(* IEC 61131-3 sources: ATCMcontrol_Engineering/src/Target/ATHW119/Libs/ATCM_IEC1131_3, 218 files *)

(* ---- ABS.st ---- *)
(*[[
    UserURL= "ATCMfile:ABS.htm"
]]*)

FUNCTION ABS : any_num
VAR_INPUT
    IN : any_num;
END_VAR

overload lreal(lreal)
inline
{
	%1
	abs_lreal
}

overload real(real)
inline
{
	%1
	abs_real
}

overload dint(dint)
inline
{
	%1
	abs_dint
}

overload int(int)
inline
{
	%1
	abs_int
}

END_FUNCTION

(* ---- ACOS.st ---- *)
FUNCTION ACOS : any_real
VAR_INPUT
    IN : any_real;
END_VAR

overload lreal(lreal) inline { STDLIB(acos_lreal) }
overload real(real)   inline { STDLIB(acos_real) }

END_FUNCTION

(* ---- add.st ---- *)
(*[[
    UserURL= "ATCMFile:ADD.htm"
]]*)

FUNCTION ADD : ANY_MAGNITUDE
VAR_INPUT
    IN1 : ANY_MAGNITUDE;
END_VAR
VAR_IN_EXT
    IN2 : ANY_MAGNITUDE;
END_VAR

inline +

END_FUNCTION

(* ---- add_time.st ---- *)
(*[[
    UserURL= "ATCMfile:ADD_TIME.htm"
]]*)

FUNCTION ADD_TIME : TIME
VAR_INPUT
    IN1 : TIME;
    IN2 : TIME;
END_VAR

inline +

END_FUNCTION

(* ---- and.st ---- *)
(*[[
    UserURL= "ATCMfile:AND.htm"
]]*)

FUNCTION AND : ANY_BIT
VAR_INPUT
    IN1 : ANY_BIT;
END_VAR
VAR_IN_EXT
    IN2 : ANY_BIT;
END_VAR

inline AND

END_FUNCTION

(* ---- ASIN.st ---- *)
FUNCTION ASIN : any_real
VAR_INPUT
    IN : any_real;
END_VAR

overload lreal(lreal) inline { STDLIB(asin_lreal) }
overload real(real) inline   { STDLIB(asin_real) }

END_FUNCTION

(* ---- ATAN.st ---- *)
FUNCTION ATAN : any_real
VAR_INPUT
    IN : any_real;
END_VAR

overload lreal(lreal) inline { STDLIB(atan_lreal) }
overload real(real)   inline { STDLIB(atan_real) }

END_FUNCTION

(* ---- bool_to_byte.st ---- *)
(*[[
    UserURL= "ATCMfile:BOOL_TO_BYTE.htm"
]]*)

FUNCTION BOOL_TO_BYTE : BYTE
VAR_INPUT
    IN : BOOL;
END_VAR

inline { VMOP(bool_to_byte) }

END_FUNCTION

(* ---- bool_to_dint.st ---- *)
(*[[
    UserURL= "ATCMfile:BOOL_TO_DINT.htm"
]]*)

FUNCTION BOOL_TO_DINT : DINT
VAR_INPUT
    IN : BOOL;
END_VAR

inline{ VMOP(bool_to_dword) }

END_FUNCTION

(* ---- bool_to_dword.st ---- *)
(*[[
    UserURL= "ATCMfile:BOOL_TO_DWORD.htm"
]]*)

FUNCTION BOOL_TO_DWORD : DWORD
VAR_INPUT
    IN : BOOL;
END_VAR

inline{ VMOP(bool_to_dword) }

END_FUNCTION

(* ---- bool_to_int.st ---- *)
(*[[
    UserURL= "ATCMfile:BOOL_TO_DINT.htm"
]]*)

FUNCTION BOOL_TO_INT : INT
VAR_INPUT
    IN : BOOL;
END_VAR

inline{ VMOP(bool_to_word) }

END_FUNCTION

(* ---- bool_to_lreal.st ---- *)
(*[[
    UserURL= "ATCMfile:BOOL_TO_LREAL.htm"
]]*)

FUNCTION BOOL_TO_LREAL : LREAL
VAR_INPUT
    IN : BOOL;
END_VAR

inline{ VMOP(BOOL_TO_LREAL) }

END_FUNCTION

(* ---- bool_to_real.st ---- *)
(*[[
    UserURL= "ATCMfile:BOOL_TO_LREAL.htm"
]]*)

FUNCTION BOOL_TO_REAL : REAL
VAR_INPUT
    IN : BOOL;
END_VAR

inline{ VMOP }

END_FUNCTION

(* ---- bool_to_string.st ---- *)
(*[[
    UserURL= "ATCMfile:BOOL_TO_WSTRING.htm"
]]*)

FUNCTION BOOL_TO_STRING : STRING
VAR_INPUT
    IN : BOOL;
END_VAR

inline{ STDLIB(bool_to_string) }

END_FUNCTION

(* ---- bool_to_udint.st ---- *)
(*[[
    UserURL= "ATCMfile:BOOL_TO_UDINT.htm"
]]*)
FUNCTION BOOL_TO_UDINT : UDINT
VAR_INPUT
    IN : BOOL;
END_VAR

inline{ VMOP }

END_FUNCTION

(* ---- bool_to_uint.st ---- *)
(*[[
    UserURL= "ATCMfile:BOOL_TO_UINT.htm"
]]*)
FUNCTION BOOL_TO_UINT : UINT
VAR_INPUT
    IN : BOOL;
END_VAR

inline{ VMOP }

END_FUNCTION

(* ---- bool_to_word.st ---- *)
(*[[
    UserURL= "ATCMfile:BOOL_TO_WORD.htm"
]]*)

FUNCTION BOOL_TO_WORD : WORD
VAR_INPUT
    IN : BOOL;
END_VAR

inline{ VMOP }

END_FUNCTION

(* ---- byte_to_bool.st ---- *)
(*[[
    UserURL= "ATCMfile:BYTE_TO_BOOL.htm"
]]*)

FUNCTION BYTE_TO_BOOL : BOOL
VAR_INPUT
    IN : BYTE;
END_VAR

inline{VMOP}

END_FUNCTION

(* ---- byte_to_dint.st ---- *)
(*[[
    UserURL= "ATCMfile:BYTE_TO_DINT.htm"
]]*)

FUNCTION BYTE_TO_DINT : DINT
VAR_INPUT
    IN : BYTE;
END_VAR

inline{ VMOP(byte_to_dword) }

END_FUNCTION

(* ---- byte_to_dword.st ---- *)
(*[[
    UserURL= "ATCMfile:BYTE_TO_DWORD.htm"
]]*)

FUNCTION BYTE_TO_DWORD : DWORD
VAR_INPUT
    IN : BYTE;
END_VAR

inline{ VMOP }

END_FUNCTION

(* ---- byte_to_int.st ---- *)
(*[[
    UserURL= "ATCMfile:BYTE_TO_DINT.htm"
]]*)

FUNCTION BYTE_TO_INT : INT
VAR_INPUT
    IN : BYTE;
END_VAR

inline{ VMOP(byte_to_word) }

END_FUNCTION

(* ---- byte_to_lreal.st ---- *)
(*[[
    UserURL= "ATCMfile:BYTE_TO_LREAL.htm"
]]*)

FUNCTION BYTE_TO_LREAL : LREAL
VAR_INPUT
    IN : BYTE;
END_VAR

inline{VMOP}

END_FUNCTION

(* ---- byte_to_real.st ---- *)
(*[[
    UserURL= "ATCMfile:BYTE_TO_LREAL.htm"
]]*)

FUNCTION BYTE_TO_REAL : REAL
VAR_INPUT
    IN : BYTE;
END_VAR

inline{VMOP}

END_FUNCTION

(* ---- byte_to_string.st ---- *)
(*[[
    UserURL= "ATCMfile:BYTE_TO_WSTRING.htm"
]]*)

FUNCTION BYTE_TO_STRING : STRING
VAR_INPUT
    IN : BYTE;
END_VAR

inline{ STDLIB(byte_to_string) }

END_FUNCTION

(* ---- byte_to_udint.st ---- *)
(*[[
    UserURL= "ATCMfile:BYTE_TO_UDINT.htm"
]]*)
FUNCTION BYTE_TO_UDINT : UDINT
VAR_INPUT
    IN : BYTE;
END_VAR

inline{ VMOP }

END_FUNCTION

(* ---- byte_to_uint.st ---- *)
(*[[
    UserURL= "ATCMfile:BYTE_TO_UINT.htm"
]]*)
FUNCTION BYTE_TO_UINT : UINT
VAR_INPUT
    IN : BYTE;
END_VAR

inline{ VMOP }

END_FUNCTION

(* ---- byte_to_word.st ---- *)
(*[[
    UserURL= "ATCMfile:BYTE_TO_WORD.htm"
]]*)

FUNCTION BYTE_TO_WORD : WORD
VAR_INPUT
    IN : BYTE;
END_VAR

inline{VMOP}

END_FUNCTION

(* ---- CONCAT.st ---- *)
FUNCTION CONCAT : ANY_STRING
VAR_INPUT
    IN1 : ANY_STRING;
END_VAR
VAR_IN_EXT
    IN2 : ANY_STRING;
END_VAR

overload STRING(STRING,STRING,...) inline { STDLIB(ConcatString) }

END_FUNCTION

(* ---- COS.st ---- *)
FUNCTION COS : any_real
VAR_INPUT
    IN : any_real;
END_VAR

overload lreal(lreal) inline { STDLIB(cos_lreal) }
overload real(real) inline   { STDLIB(cos_real) }

END_FUNCTION

(* ---- DELETE.st ---- *)
FUNCTION DELETE : ANY_STRING
VAR_INPUT
    IN : ANY_STRING;
    L : ANY_INT;
    P : ANY_INT;
END_VAR

overload STRING(STRING,         INT,         INT) inline{ STDLIB(DeleteString_int)}
overload STRING(STRING, DINT to INT, DINT to INT) inline{ STDLIB(DeleteString_int)}

END_FUNCTION

(* ---- dint_to_bool.st ---- *)
(*[[
    UserURL= "ATCMfile:DINT_TO_BOOL.htm"
]]*)

FUNCTION DINT_TO_BOOL : BOOL
VAR_INPUT
    IN : DINT;
END_VAR

inline{ VMOP(dword_to_bool) }

END_FUNCTION

(* ---- dint_to_byte.st ---- *)
(*[[
    UserURL= "ATCMfile:DINT_TO_BYTE.htm"
]]*)

FUNCTION DINT_TO_BYTE : BYTE
VAR_INPUT
    IN : DINT;
END_VAR

inline{ VMOP }

END_FUNCTION

(* ---- dint_to_dword.st ---- *)
(*[[
    UserURL= "ATCMfile:DINT_TO_DWORD.htm"
]]*)

FUNCTION DINT_TO_DWORD : DWORD
VAR_INPUT
    IN : DINT;
END_VAR

inline{NOOP}

END_FUNCTION

(* ---- dint_to_int.st ---- *)
(*[[
    UserURL= "ATCMfile:DINT_TO_LINT.htm"
]]*)

FUNCTION DINT_TO_INT : INT
VAR_INPUT
    IN : DINT;
END_VAR

inline{VMOP}

END_FUNCTION

(* ---- dint_to_lreal.st ---- *)
(*[[
    UserURL= "ATCMfile:DINT_TO_LREAL.htm"
]]*)

FUNCTION DINT_TO_LREAL : LREAL
VAR_INPUT
    IN : DINT;
END_VAR

inline{VMOP}

END_FUNCTION

(* ---- dint_to_real.st ---- *)
(*[[
    UserURL= "ATCMfile:DINT_TO_LREAL.htm"
]]*)

FUNCTION DINT_TO_REAL : REAL
VAR_INPUT
    IN : DINT;
END_VAR

inline{VMOP}

END_FUNCTION

(* ---- dint_to_string.st ---- *)
(*[[
    UserURL= "ATCMfile:DINT_TO_WSTRING.htm"
]]*)

FUNCTION DINT_TO_STRING : STRING
VAR_INPUT
    IN : DINT;
END_VAR

inline{ STDLIB(dint_to_string) }

END_FUNCTION

(* ---- dint_to_time.st ---- *)
(*[[
    UserURL= "ATCMfile:DINT_TO_TIME.htm"
]]*)

FUNCTION DINT_TO_TIME : TIME
VAR_INPUT
    IN : DINT;
END_VAR

inline { %1 }

END_FUNCTION

(* ---- dint_to_udint.st ---- *)
(*[[
    UserURL= "ATCMfile:DINT_TO_UDINT.htm"
]]*)
FUNCTION DINT_TO_UDINT : UDINT
VAR_INPUT
    IN : DINT;
END_VAR

inline{NOOP}

END_FUNCTION

(* ---- dint_to_uint.st ---- *)
(*[[
    UserURL= "ATCMfile:DINT_TO_UINT.htm"
]]*)
FUNCTION DINT_TO_UINT : UINT
VAR_INPUT
    IN : DINT;
END_VAR

inline{ VMOP }

END_FUNCTION

(* ---- dint_to_word.st ---- *)
(*[[
    UserURL= "ATCMfile:DINT_TO_WORD.htm"
]]*)

FUNCTION DINT_TO_WORD : WORD
VAR_INPUT
    IN : DINT;
END_VAR

inline{VMOP}

END_FUNCTION

(* ---- div.st ---- *)
(*[[
    UserURL= "ATCMfile:DIV.htm"
]]*)

FUNCTION DIV : ANY_NUM
VAR_INPUT
    IN1: ANY_NUM;
    IN2: ANY_NUM;
END_VAR

inline /

END_FUNCTION

(* ---- divtime.st ---- *)
(*[[
    UserURL= "ATCMfile:DIVTIME.htm"
]]*)

FUNCTION DIVTIME : TIME
VAR_INPUT
    IN1 : TIME;
    IN2 : ANY_NUM;
END_VAR

overload TIME(TIME,INT)
inline
{
    %1
    %2
    int_to_dint
    div_dint
}

overload TIME(TIME,DINT)
inline
{
    %1
    %2
    div_dint
}

overload TIME(TIME,REAL)
inline
{
    %1
    dint_to_real
    %2
    div_real
    real_to_dint
}

overload TIME(TIME,LREAL)
inline
{
    %1
    dint_to_lreal
    %2
    div_lreal
    lreal_to_dint
}

END_FUNCTION

(* ---- dword_to_bool.st ---- *)
(*[[
    UserURL= "ATCMfile:DWORD_TO_BOOL.htm"
]]*)

FUNCTION DWORD_TO_BOOL : BOOL
VAR_INPUT
    IN : DWORD;
END_VAR

inline{VMOP}

END_FUNCTION

(* ---- dword_to_byte.st ---- *)
(*[[
    UserURL= "ATCMfile:DWORD_TO_BYTE.htm"
]]*)

FUNCTION DWORD_TO_BYTE : BYTE
VAR_INPUT
    IN : DWORD;
END_VAR

inline{VMOP}

END_FUNCTION

(* ---- dword_to_dint.st ---- *)
(*[[
    UserURL= "ATCMfile:DWORD_TO_DINT.htm"
]]*)

FUNCTION DWORD_TO_DINT : DINT
VAR_INPUT
    IN : DWORD;
END_VAR

inline{VMOP}

END_FUNCTION

(* ---- dword_to_int.st ---- *)
(*[[
    UserURL= "ATCMfile:DWORD_TO_LINT.htm"
]]*)

FUNCTION DWORD_TO_INT : INT
VAR_INPUT
    IN : DWORD;
END_VAR

inline{VMOP}

END_FUNCTION

(* ---- dword_to_lreal.st ---- *)
(*[[
    UserURL= "ATCMfile:DWORD_TO_LREAL.htm"
]]*)

FUNCTION DWORD_TO_LREAL : LREAL
VAR_INPUT
    IN : DWORD;
END_VAR

inline{VMOP}

END_FUNCTION

(* ---- dword_to_lword.st ---- *)
(*[[
    UserURL= "ATCMfile:DWORD_TO_LWORD.htm"
]]*)

FUNCTION DWORD_TO_LWORD : LWORD
VAR_INPUT
    IN : DWORD;
END_VAR

inline{VMOP}

END_FUNCTION

(* ---- dword_to_real.st ---- *)
(*[[
    UserURL= "ATCMfile:DWORD_TO_LREAL.htm"
]]*)

FUNCTION DWORD_TO_REAL : REAL
VAR_INPUT
    IN : DWORD;
END_VAR

inline{VMOP}

END_FUNCTION

(* ---- dword_to_string.st ---- *)
(*[[
    UserURL= "ATCMfile:DWORD_TO_WSTRING.htm"
]]*)

FUNCTION DWORD_TO_STRING : STRING
VAR_INPUT
    IN : DWORD;
END_VAR

inline{ STDLIB(dword_to_string) }

END_FUNCTION

(* ---- dword_to_udint.st ---- *)
(*[[
    UserURL= "ATCMfile:DWORD_TO_UDINT.htm"
]]*)
FUNCTION DWORD_TO_UDINT : UDINT
VAR_INPUT
    IN : DWORD;
END_VAR

inline{NOOP}

END_FUNCTION

(* ---- dword_to_uint.st ---- *)
(*[[
    UserURL= "ATCMfile:DWORD_TO_UINT.htm"
]]*)
FUNCTION DWORD_TO_UINT : UINT
VAR_INPUT
    IN : DWORD;
END_VAR

inline{ VMOP }

END_FUNCTION

(* ---- dword_to_word.st ---- *)
(*[[
    UserURL= "ATCMfile:DWORD_TO_WORD.htm"
]]*)

FUNCTION DWORD_TO_WORD : WORD
VAR_INPUT
    IN : DWORD;
END_VAR

inline{VMOP(dword_to_uint)}

END_FUNCTION

(* ---- eq.st ---- *)
(*[[
    UserURL= "ATCMfile:EQ.htm"
]]*)

FUNCTION EQ : BOOL
VAR_INPUT
    IN1 : ANY_ELEMENTARY;
END_VAR
VAR_IN_EXT
    IN2 : ANY_ELEMENTARY;
END_VAR

inline =

END_FUNCTION

(* ---- EXP.st ---- *)
FUNCTION EXP : any_real
VAR_INPUT
    IN : any_real;
END_VAR

overload lreal(lreal) inline { STDLIB(exp_lreal) }
overload real(real)   inline { STDLIB(exp_real) }

END_FUNCTION

(* ---- expt.st ---- *)
(*[[
    UserURL= "ATCMfile:EXPT.htm"
]]*)

FUNCTION EXPT : ANY_REAL
VAR_INPUT
    IN1: ANY_REAL;
    IN2: ANY_NUM;
END_VAR

overload REAL(REAL,DINT)    inline
{
    %1
    %2
    pow_real_dint
}
overload REAL(REAL,INT)     inline
{
    %1
    %2
    pow_real_int
}
overload LREAL(LREAL,DINT)  inline
{
    %1
    %2
    pow_lreal_dint
}
overload LREAL(LREAL,INT)   inline
{
    %1
    %2
    pow_lreal_int
}
overload REAL(REAL,REAL)    inline
{
    %1
    %2
    pow_real_real
}
overload LREAL(LREAL,LREAL) inline
{
    %1
    %2
    pow_lreal_lreal
}
overload REAL(REAL,LREAL)   inline
{
    %1
    real_to_lreal
    %2
    pow_lreal_lreal
    lreal_to_real
}
overload LREAL(LREAL,REAL)  inline
{
    %1
    %2
    real_to_lreal
    pow_lreal_lreal
}

END_FUNCTION

(* ---- FIND.st ---- *)
FUNCTION FIND : ANY_INT
VAR_INPUT
    IN1 : ANY_STRING;
    IN2 : ANY_STRING;
END_VAR

overload INT        (STRING, STRING) inline{ STDLIB(FindString_int) }
overload INT to DINT(STRING, STRING) inline{ STDLIB(FindString_int) }

END_FUNCTION

(* ---- ge.st ---- *)
(*[[
    UserURL= "ATCMfile:GE.htm"
]]*)

FUNCTION GE : BOOL
VAR_INPUT
    IN1 : ANY_ELEMENTARY;
END_VAR
VAR_IN_EXT
    IN2 : ANY_ELEMENTARY;
END_VAR

inline >=

END_FUNCTION

(* ---- gt.st ---- *)
(*[[
    UserURL= "ATCMfile:GT.htm"
]]*)

FUNCTION GT : BOOL
VAR_INPUT
    IN1 : ANY_ELEMENTARY;
END_VAR
VAR_IN_EXT
    IN2 : ANY_ELEMENTARY;
END_VAR

inline >

END_FUNCTION

(* ---- INSERT.st ---- *)
FUNCTION INSERT : ANY_STRING
VAR_INPUT
    IN1 : ANY_STRING;
    IN2 : ANY_STRING;
    P : ANY_INT;
END_VAR

overload STRING(STRING, STRING,         INT) inline{ STDLIB(InsertString_int)}
overload STRING(STRING, STRING, DINT to INT) inline{ STDLIB(InsertString_int)}

END_FUNCTION

(* ---- int_to_bool.st ---- *)
(*[[
    UserURL= "ATCMfile:DINT_TO_BOOL.htm"
]]*)

FUNCTION INT_TO_BOOL : BOOL
VAR_INPUT
    IN : INT;
END_VAR

inline{VMOP(WORD_TO_BOOL)}

END_FUNCTION

(* ---- int_to_byte.st ---- *)
(*[[
    UserURL= "ATCMfile:DINT_TO_BYTE.htm"
]]*)

FUNCTION INT_TO_BYTE : BYTE
VAR_INPUT
    IN : INT;
END_VAR

inline{VMOP(word_to_byte)}

END_FUNCTION

(* ---- int_to_dint.st ---- *)
(*[[
    UserURL= "ATCMfile:DINT_TO_LINT.htm"
]]*)

FUNCTION INT_TO_DINT : DINT
VAR_INPUT
    IN : INT;
END_VAR

inline{VMOP}

END_FUNCTION

(* ---- int_to_dword.st ---- *)
(*[[
    UserURL= "ATCMfile:DINT_TO_DWORD.htm"
]]*)

FUNCTION INT_TO_DWORD : DWORD
VAR_INPUT
    IN : INT;
END_VAR

inline{VMOP(int_to_dword)}

END_FUNCTION

(* ---- int_to_lint.st ---- *)
(*[[
    UserURL= "ATCMfile:DINT_TO_LINT.htm"
]]*)

FUNCTION INT_TO_LINT : LINT
VAR_INPUT
    IN : INT;
END_VAR

inline{VMOP}

END_FUNCTION

(* ---- int_to_lreal.st ---- *)
(*[[
    UserURL= "ATCMfile:DINT_TO_LREAL.htm"
]]*)

FUNCTION INT_TO_LREAL : LREAL
VAR_INPUT
    IN : INT;
END_VAR

inline{VMOP}

END_FUNCTION

(* ---- int_to_real.st ---- *)
(*[[
    UserURL= "ATCMfile:DINT_TO_LREAL.htm"
]]*)

FUNCTION INT_TO_REAL : REAL
VAR_INPUT
    IN : INT;
END_VAR

inline{VMOP}

END_FUNCTION

(* ---- int_to_string.st ---- *)
(*[[
    UserURL= "ATCMfile:DINT_TO_WSTRING.htm"
]]*)

FUNCTION INT_TO_STRING : STRING
VAR_INPUT
    IN : INT;
END_VAR

inline{ STDLIB(int_to_string) }

END_FUNCTION

(* ---- int_to_time.st ---- *)
(*[[
    UserURL= "ATCMfile:DINT_TO_TIME.htm"
]]*)

FUNCTION INT_TO_TIME : TIME
VAR_INPUT
    IN : INT;
END_VAR

inline
{
	%1
	int_to_dint
}

END_FUNCTION

(* ---- int_to_udint.st ---- *)
(*[[
    UserURL= "ATCMfile:INT_TO_UDINT.htm"
]]*)
FUNCTION INT_TO_UDINT : UDINT
VAR_INPUT
    IN : INT;
END_VAR

inline{ VMOP }

END_FUNCTION

(* ---- int_to_uint.st ---- *)
(*[[
    UserURL= "ATCMfile:INT_TO_UINT.htm"
]]*)
FUNCTION INT_TO_UINT : UINT
VAR_INPUT
    IN : INT;
END_VAR

inline{NOOP}

END_FUNCTION

(* ---- int_to_word.st ---- *)
(*[[
    UserURL= "ATCMfile:DINT_TO_WORD.htm"
]]*)

FUNCTION INT_TO_WORD : WORD
VAR_INPUT
    IN : INT;
END_VAR

inline{NOOP}

END_FUNCTION

(* ---- le.st ---- *)
(*[[
    UserURL= "ATCMfile:LE.htm"
]]*)

FUNCTION LE : BOOL
VAR_INPUT
    IN1 : ANY_ELEMENTARY;
END_VAR
VAR_IN_EXT
    IN2 : ANY_ELEMENTARY;
END_VAR

inline <=

END_FUNCTION

(* ---- LEFT.st ---- *)
FUNCTION LEFT : ANY_STRING
VAR_INPUT
    IN : ANY_STRING;
    L : ANY_INT;
END_VAR

overload STRING(STRING, INT)          inline{ STDLIB(LeftString_int) }
overload STRING(STRING, DINT to INT)  inline{ STDLIB(LeftString_int) }

END_FUNCTION

(* ---- LEN.st ---- *)
FUNCTION LEN : ANY_INT
VAR_INPUT
    IN : STRING;
END_VAR

overload INT        (STRING) inline { STDLIB(strlen_int) }
overload INT to DINT(STRING) inline { STDLIB(strlen_int) }

END_FUNCTION

(* ---- limit.st ---- *)
(*[[
    UserURL= "ATCMfile:LIMIT.htm"
]]*)

FUNCTION LIMIT : ANY_ELEMENTARY
VAR_INPUT
    MN : ANY_ELEMENTARY;
    IN : ANY_ELEMENTARY;
    MX : ANY_ELEMENTARY;
END_VAR

overload BOOL(BOOL,BOOL,BOOL) inline
{
    %2
    %1
    or_bool
    %3
    and_bool
}
overload BYTE(BYTE, BYTE, BYTE) inline
{
    %2
    %1
    lt_byte
    jmpcn L1%u
    %1
    jmp Lend%u
:L1%u
    %2
    %3
    gt_byte
    jmpcn L2%u
    %3
    jmp Lend%u
:L2%u
    %2
:Lend%u
}
overload WORD(WORD, WORD, WORD) inline
{
    %2
    %1
    lt_word
    jmpcn L1%u
    %1
    jmp Lend%u
:L1%u
    %2
    %3
    gt_word
    jmpcn L2%u
    %3
    jmp Lend%u
:L2%u
    %2
:Lend%u
}
overload DWORD(DWORD, DWORD, DWORD) inline
{
    %2
    %1
    lt_dword
    jmpcn L1%u
    %1
    jmp Lend%u
:L1%u
    %2
    %3
    gt_dword
    jmpcn L2%u
    %3
    jmp Lend%u
:L2%u
    %2
:Lend%u
}
overload INT(INT, INT, INT) inline
{
    %2
    %1
    lt_int
    jmpcn L1%u
    %1
    jmp Lend%u
:L1%u
    %2
    %3
    gt_int
    jmpcn L2%u
    %3
    jmp Lend%u
:L2%u
    %2
:Lend%u
}
overload DINT|TIME(DINT|TIME, DINT|TIME, DINT|TIME) inline
{
    %2
    %1
    lt_dint
    jmpcn L1%u
    %1
    jmp Lend%u
:L1%u
    %2
    %3
    gt_dint
    jmpcn L2%u
    %3
    jmp Lend%u
:L2%u
    %2
:Lend%u
}
overload REAL(REAL,REAL,REAL) inline
{
    %2
    %1
    lt_real
    jmpcn L1%u
    %1
    jmp Lend%u
:L1%u
    %2
    %3
    gt_real
    jmpcn L2%u
    %3
    jmp Lend%u
:L2%u
    %2
:Lend%u
}

overload LREAL(LREAL,LREAL,LREAL) inline
{
    %2
    %1
    lt_lreal
    jmpcn L1%u
    %1
    jmp Lend%u
:L1%u
    %2
    %3
    gt_lreal
    jmpcn L2%u
    %3
    jmp Lend%u
:L2%u
    %2
:Lend%u
}

overload STRING(STRING, STRING, STRING) inline
{
    %2
    %1
    lt_string
    jmpcn L1%u
    %1
    jmp Lend%u
:L1%u
    %2
    %3
    gt_string
    jmpcn L2%u
    %3
    jmp Lend%u
:L2%u
    %2
:Lend%u
}

END_FUNCTION

(* ---- lint_to_bool.st ---- *)
(*[[
    UserURL= "ATCMfile:LINT_TO_BOOL.htm"
]]*)

FUNCTION LINT_TO_BOOL : BOOL
VAR_INPUT
    IN : LINT;
END_VAR

inline{%1==0l?false:true}

END_FUNCTION

(* ---- lint_to_byte.st ---- *)
(*[[
    UserURL= "ATCMfile:LINT_TO_BYTE.htm"
]]*)

FUNCTION LINT_TO_BYTE : BYTE
VAR_INPUT
    IN : LINT;
END_VAR

inline{(int)%1&0xff}

END_FUNCTION

(* ---- lint_to_dint.st ---- *)
(*[[
    UserURL= "ATCMfile:LINT_TO_DINT.htm"
]]*)

FUNCTION LINT_TO_DINT : DINT
VAR_INPUT
    IN : LINT;
END_VAR

inline{(int)%1}

END_FUNCTION

(* ---- lint_to_dword.st ---- *)
(*[[
    UserURL= "ATCMfile:LINT_TO_DWORD.htm"
]]*)

FUNCTION LINT_TO_DWORD : DWORD
VAR_INPUT
    IN : LINT;
END_VAR

inline{(int)%1}

END_FUNCTION

(* ---- lint_to_int.st ---- *)
(*[[
    UserURL= "ATCMfile:LINT_TO_DINT.htm"
]]*)

FUNCTION LINT_TO_INT : INT
VAR_INPUT
    IN : LINT;
END_VAR

inline{(int)%1}

END_FUNCTION

(* ---- lint_to_lreal.st ---- *)
(*[[
    UserURL= "ATCMfile:LINT_TO_LREAL.htm"
]]*)

FUNCTION LINT_TO_LREAL : LREAL
VAR_INPUT
    IN : LINT;
END_VAR

inline{(double)%1}

END_FUNCTION

(* ---- lint_to_lword.st ---- *)
(*[[
    UserURL= "ATCMfile:LINT_TO_LWORD.htm"
]]*)

FUNCTION LINT_TO_LWORD : LWORD
VAR_INPUT
    IN : LINT;
END_VAR

inline{%1}

END_FUNCTION

(* ---- lint_to_real.st ---- *)
(*[[
    UserURL= "ATCMfile:LINT_TO_LREAL.htm"
]]*)

FUNCTION LINT_TO_REAL : REAL
VAR_INPUT
    IN : LINT;
END_VAR

inline{(double)%1}

END_FUNCTION

(* ---- lint_to_string.st ---- *)
(*[[
    UserURL= "ATCMfile:LINT_TO_WSTRING.htm"
]]*)

FUNCTION LINT_TO_STRING : STRING
VAR_INPUT
    IN : LINT;
END_VAR

inline{java.lang.Long.toString(%1)}

END_FUNCTION

(* ---- lint_to_time.st ---- *)
(*[[
    UserURL= "ATCMfile:LINT_TO_TIME.htm"
]]*)

FUNCTION LINT_TO_TIME : TIME
VAR_INPUT
    IN : LINT;
END_VAR

inline{%1}

END_FUNCTION

(* ---- lint_to_word.st ---- *)
(*[[
    UserURL= "ATCMfile:LINT_TO_WORD.htm"
]]*)

FUNCTION LINT_TO_WORD : WORD
VAR_INPUT
    IN : LINT;
END_VAR

inline{(int)%1&0xffff}

END_FUNCTION

(* ---- LN.st ---- *)
FUNCTION LN : any_real
VAR_INPUT
    IN : any_real;
END_VAR

overload lreal(lreal) inline { STDLIB(log_lreal) }
overload real(real)   inline { STDLIB(log_real) }

END_FUNCTION

(* ---- LOG.st ---- *)
FUNCTION LOG : any_real
VAR_INPUT
    IN : any_real;
END_VAR

overload lreal(lreal) inline { STDLIB(log10_lreal) }
overload real(real)   inline { STDLIB(log10_real) }

END_FUNCTION

(* ---- lreal_to_bool.st ---- *)
(*[[
    UserURL= "ATCMfile:LREAL_TO_BOOL.htm"
]]*)

FUNCTION LREAL_TO_BOOL : BOOL
VAR_INPUT
    IN : LREAL;
END_VAR

inline{VMOP}

END_FUNCTION

(* ---- lreal_to_byte.st ---- *)
(*[[
    UserURL= "ATCMfile:LREAL_TO_BYTE.htm"
]]*)

FUNCTION LREAL_TO_BYTE : BYTE
VAR_INPUT
    IN : LREAL;
END_VAR

inline{VMOP}

END_FUNCTION

(* ---- lreal_to_dint.st ---- *)
(*[[
    UserURL= "ATCMfile:LREAL_TO_DINT.htm"
]]*)

FUNCTION LREAL_TO_DINT : DINT
VAR_INPUT
    IN : LREAL;
END_VAR

inline{VMOP}

END_FUNCTION

(* ---- lreal_to_dword.st ---- *)
(*[[
    UserURL= "ATCMfile:LREAL_TO_DWORD.htm"
]]*)

FUNCTION LREAL_TO_DWORD : DWORD
VAR_INPUT
    IN : LREAL;
END_VAR

inline{VMOP}

END_FUNCTION

(* ---- lreal_to_int.st ---- *)
(*[[
    UserURL= "ATCMfile:LREAL_TO_LINT.htm"
]]*)

FUNCTION LREAL_TO_INT : INT
VAR_INPUT
    IN : LREAL;
END_VAR

inline{VMOP}

END_FUNCTION

(* ---- lreal_to_lint.st ---- *)
(*[[
    UserURL= "ATCMfile:LREAL_TO_LINT.htm"
]]*)

FUNCTION LREAL_TO_LINT : LINT
VAR_INPUT
    IN : LREAL;
END_VAR

inline{VMOP(not_yet_implem)}

END_FUNCTION

(* ---- lreal_to_lword.st ---- *)
(*
 * Note:
 *  LREAL_TO_LWORD(x) is the same as
 *  LINT_TO_LWORD(LREAL_TO_LINT(x))
 *
 *  e.g.  LREAL_TO_LWORD(-1.0E0) = 16#ffffffffffffffff;
 *)

FUNCTION LREAL_TO_LWORD : LWORD
VAR_INPUT
    IN : LREAL;
END_VAR

inline{VMOP(not_yet_implem)}

END_FUNCTION

(* ---- lreal_to_real.st ---- *)
(*[[
    UserURL= "ATCMfile:LREAL_TO_TIME.htm"
]]*)

FUNCTION LREAL_TO_REAL : REAL
VAR_INPUT
    IN : LREAL;
END_VAR

inline{VMOP}

END_FUNCTION

(* ---- lreal_to_string.st ---- *)
(*[[
    UserURL= "ATCMfile:LREAL_TO_WSTRING.htm"
]]*)

FUNCTION LREAL_TO_STRING : STRING
VAR_INPUT
    IN : LREAL;
END_VAR

inline{ STDLIB(lreal_to_string)}

END_FUNCTION

(* ---- lreal_to_time.st ---- *)
(*[[
    UserURL= "ATCMfile:LREAL_TO_TIME.htm"
]]*)

FUNCTION LREAL_TO_TIME : TIME
VAR_INPUT
    IN : LREAL;
END_VAR

inline
{
    %1
	lreal_to_dint
}

END_FUNCTION

(* ---- lreal_to_udint.st ---- *)
(*[[
    UserURL= "ATCMfile:LREAL_TO_UDINT.htm"
]]*)
FUNCTION LREAL_TO_UDINT : UDINT
VAR_INPUT
    IN : LREAL;
END_VAR

inline{ VMOP }

END_FUNCTION

(* ---- lreal_to_uint.st ---- *)
(*[[
    UserURL= "ATCMfile:LREAL_TO_UINT.htm"
]]*)
FUNCTION LREAL_TO_UINT : UINT
VAR_INPUT
    IN : LREAL;
END_VAR

inline{ VMOP }

END_FUNCTION

(* ---- lreal_to_word.st ---- *)
(*[[
    UserURL= "ATCMfile:LREAL_TO_WORD.htm"
]]*)

FUNCTION LREAL_TO_WORD : WORD
VAR_INPUT
    IN : LREAL;
END_VAR

inline{VMOP}

END_FUNCTION

(* ---- lt.st ---- *)
(*[[
    UserURL= "ATCMfile:LT.htm"
]]*)

FUNCTION LT : BOOL
VAR_INPUT
    IN1 : ANY_ELEMENTARY;
END_VAR
VAR_IN_EXT
    IN2 : ANY_ELEMENTARY;
END_VAR

inline <

END_FUNCTION

(* ---- lword_to_bool.st ---- *)
(*[[
    UserURL= "ATCMfile:LWORD_TO_BOOL.htm"
]]*)

FUNCTION LWORD_TO_BOOL : BOOL
VAR_INPUT
    IN : LWORD;
END_VAR

inline{%1==0l?false:true}

END_FUNCTION

(* ---- lword_to_byte.st ---- *)
(*[[
    UserURL= "ATCMfile:LWORD_TO_BYTE.htm"
]]*)

FUNCTION LWORD_TO_BYTE : BYTE
VAR_INPUT
    IN : LWORD;
END_VAR

inline{(int)%1&0xff}

END_FUNCTION

(* ---- lword_to_dint.st ---- *)
(*[[
    UserURL= "ATCMfile:LWORD_TO_DINT.htm"
]]*)

FUNCTION LWORD_TO_DINT : DINT
VAR_INPUT
    IN : LWORD;
END_VAR

inline{(int)%1}

END_FUNCTION

(* ---- lword_to_dword.st ---- *)
(*[[
    UserURL= "ATCMfile:LWORD_TO_DWORD.htm"
]]*)

FUNCTION LWORD_TO_DWORD : DWORD
VAR_INPUT
    IN : LWORD;
END_VAR

inline{(int)%1}

END_FUNCTION

(* ---- lword_to_int.st ---- *)
(*[[
    UserURL= "ATCMfile:LWORD_TO_DINT.htm"
]]*)

FUNCTION LWORD_TO_INT : INT
VAR_INPUT
    IN : LWORD;
END_VAR

inline{(int)%1}

END_FUNCTION

(* ---- lword_to_lint.st ---- *)
(*[[
    UserURL= "ATCMfile:LWORD_TO_LINT.htm"
]]*)

FUNCTION LWORD_TO_LINT : LINT
VAR_INPUT
    IN : LWORD;
END_VAR

inline{%1}

END_FUNCTION

(* ---- lword_to_lreal.st ---- *)
(*
 * Note:
 *  LWORD_TO_LREAL(x) is the same as
 *  LINT_TO_LREAL(LWORD_TO_LINT(x))
 *
 *  e.g.  LWORD_TO_LREAL(16#ffffffffffffffff) = -1.0E0
 *)
FUNCTION LWORD_TO_LREAL : LREAL
VAR_INPUT
    IN : LWORD;
END_VAR

inline{(double)%1}

END_FUNCTION

(* ---- lword_to_real.st ---- *)
(*
 * Note:
 *  LWORD_TO_LREAL(x) is the same as
 *  LINT_TO_LREAL(LWORD_TO_LINT(x))
 *
 *  e.g.  LWORD_TO_LREAL(16#ffffffffffffffff) = -1.0E0
 *)
FUNCTION LWORD_TO_REAL : REAL
VAR_INPUT
    IN : LWORD;
END_VAR

inline{(double)%1}

END_FUNCTION

(* ---- lword_to_string.st ---- *)
(*[[
    UserURL= "ATCMfile:LWORD_TO_WSTRING.htm"
]]*)

FUNCTION LWORD_TO_STRING : STRING
VAR_INPUT
    IN : LWORD;
END_VAR

inline{ STDLIB(not yet implemented) }

END_FUNCTION

(* ---- lword_to_word.st ---- *)
(*[[
    UserURL= "ATCMfile:LWORD_TO_WORD.htm"
]]*)

FUNCTION LWORD_TO_WORD : WORD
VAR_INPUT
    IN : LWORD;
END_VAR

inline{(int)%1&0xffff}

END_FUNCTION

(* ---- max.st ---- *)
(*[[
]]*)

FUNCTION MAX : ANY_ELEMENTARY
VAR_INPUT
    IN1 : ANY_ELEMENTARY;
END_VAR
VAR_IN_EXT
    IN2 : ANY_ELEMENTARY;
END_VAR

overload BOOL(BOOL,BOOL) inline
{
    %1
    %2
    or_bool
}
overload BYTE(BYTE,BYTE) inline
{
    %1
    %2
    gt_byte
    jmpcn L1%u
    %1
    jmp Lend%u
:L1%u
    %2
:Lend%u
}
overload WORD(WORD,WORD) inline
{
    %1
    %2
    gt_word
    jmpcn L1%u
    %1
    jmp Lend%u
:L1%u
    %2
:Lend%u
}
overload DWORD(DWORD,DWORD) inline
{
    %1
    %2
    gt_dword
    jmpcn L1%u
    %1
    jmp Lend%u
:L1%u
    %2
:Lend%u
}
overload INT(INT,INT) inline
{
    %1
    %2
    gt_int
    jmpcn L1%u
    %1
    jmp Lend%u
:L1%u
    %2
:Lend%u
}
overload DINT|TIME(DINT|TIME,DINT|TIME) inline
{
    %1
    %2
    gt_dint
    jmpcn L1%u
    %1
    jmp Lend%u
:L1%u
    %2
:Lend%u
}
overload REAL(REAL,REAL) inline
{
    %1
    %2
    gt_real
    jmpcn L1%u
    %1
    jmp Lend%u
:L1%u
    %2
:Lend%u
}
overload LREAL(LREAL,LREAL) inline
{
    %1
    %2
    gt_lreal
    jmpcn L1%u
    %1
    jmp Lend%u
:L1%u
    %2
:Lend%u
}
overload STRING(STRING,STRING) inline
{
    %1
    %2
    gt_string
    jmpcn L1%u
    %1
    jmp Lend%u
:L1%u
    %2
:Lend%u
}

(*
TODO implement extensible funs in interpreter
overload BOOL(BOOL, BOOL, ... )                        inline{ STDLIB(max_bool) }
overload BYTE(BYTE,BYTE, ... )                         inline{ STDLIB(max_byte) }
overload WORD(WORD,WORD, ... )                         inline{ STDLIB(max_word) }
overload DWORD(DWORD, DWORD, ... )                     inline{ STDLIB(max_dword) }

overload INT(INT,INT, ... )                            inline{ STDLIB(max_int) }
overload DINT(DINT,DINT, ... )                         inline{ STDLIB(max_dint) }

overload REAL(REAL,REAL, ... )                         inline{ STDLIB(max_real) }
overload LREAL(LREAL,LREAL, ... )                      inline{ STDLIB(max_lreal) }

overload TIME(TIME,TIME, ...)                          inline{ STDLIB(max_udint) }
overload STRING(STRING, STRING, ... )                  inline{ STDLIB(max_string) }
*)

END_FUNCTION

(* ---- MID.st ---- *)
FUNCTION MID : ANY_STRING
VAR_INPUT
    IN : ANY_STRING;
    L : ANY_INT;
    P : ANY_INT;
END_VAR

overload STRING(STRING,         INT,         INT) inline{ STDLIB(MidString_int) }
overload STRING(STRING, DINT to INT, DINT to INT) inline{ STDLIB(MidString_int) }

END_FUNCTION

(* ---- MIN.st ---- *)
FUNCTION MIN : ANY_ELEMENTARY
VAR_INPUT
    IN1 : ANY_ELEMENTARY;
END_VAR
VAR_IN_EXT
    IN2 : ANY_ELEMENTARY;
END_VAR

overload BOOL(BOOL,BOOL) inline
{
    %1
    %2
    and_bool
}
overload BYTE(BYTE,BYTE) inline
{
    %1
    %2
    lt_byte
    jmpcn L1%u
    %1
    jmp Lend%u
:L1%u
    %2
:Lend%u
}
overload WORD(WORD,WORD) inline
{
    %1
    %2
    lt_word
    jmpcn L1%u
    %1
    jmp Lend%u
:L1%u
    %2
:Lend%u
}
overload DWORD(DWORD,DWORD) inline
{
    %1
    %2
    lt_dword
    jmpcn L1%u
    %1
    jmp Lend%u
:L1%u
    %2
:Lend%u
}
overload INT(INT,INT) inline
{
    %1
    %2
    lt_int
    jmpcn L1%u
    %1
    jmp Lend%u
:L1%u
    %2
:Lend%u
}
overload DINT|TIME(DINT|TIME,DINT|TIME) inline
{
    %1
    %2
    lt_dint
    jmpcn L1%u
    %1
    jmp Lend%u
:L1%u
    %2
:Lend%u
}
overload REAL(REAL,REAL) inline
{
    %1
    %2
    lt_real
    jmpcn L1%u
    %1
    jmp Lend%u
:L1%u
    %2
:Lend%u
}
overload LREAL(LREAL,LREAL) inline
{
    %1
    %2
    lt_lreal
    jmpcn L1%u
    %1
    jmp Lend%u
:L1%u
    %2
:Lend%u
}

overload STRING(STRING,STRING) inline
{
    %1
    %2
    lt_string
    jmpcn L1%u
    %1
    jmp Lend%u
:L1%u
    %2
:Lend%u
}

(*
TODO implement extensible funs in interpreter
overload BOOL(BOOL, BOOL, ... )                        inline{ STDLIB(min_bool) }
overload BYTE(BYTE,BYTE, ... )                         inline{ STDLIB(min_byte) }
overload WORD(WORD,WORD, ... )                         inline{ STDLIB(min_word) }
overload DWORD(DWORD, DWORD, ... )                     inline{ STDLIB(min_dword) }

overload INT(INT,INT, ... )                            inline{ STDLIB(min_int) }
overload DINT(DINT,DINT, ... )                         inline{ STDLIB(min_dint) }

overload REAL(REAL,REAL, ... )                         inline{ STDLIB(min_real) }
overload LREAL(LREAL,LREAL, ... )                      inline{ STDLIB(min_lreal) }

overload TIME(TIME,TIME, ...)                          inline{ STDLIB(min_udint) }
overload STRING(STRING, STRING, ... )                  inline{ STDLIB(min_string) }
*)

END_FUNCTION

(* ---- mod.st ---- *)
(*[[
    UserURL= "ATCMfile:MOD.htm"
]]*)

FUNCTION MOD : ANY_INT
VAR_INPUT
    IN1: ANY_INT;
    IN2: ANY_INT;
END_VAR

inline MOD

END_FUNCTION

(* ---- move.st ---- *)
FUNCTION MOVE: ANY
VAR_INPUT
    In: ANY;
END_VAR

inline :=

END_FUNCTION

(* ---- mul.st ---- *)
(*[[
    UserURL= "ATCMfile:MUL.htm"
]]*)

FUNCTION MUL : ANY_NUM
VAR_INPUT
    IN1 : ANY_NUM;
END_VAR
VAR_IN_EXT
    IN2 : ANY_NUM;
END_VAR

inline *

END_FUNCTION

(* ---- multime.st ---- *)
(*[[
    UserURL= "ATCMfile:MULTIME.htm"
]]*)

FUNCTION MULTIME : TIME
VAR_INPUT
    IN1 : TIME;
    IN2 : ANY_NUM;
END_VAR

overload TIME(TIME,INT)
inline
{
    %1
    %2
    int_to_dint
    mul_dint
}

overload TIME(TIME,DINT)
inline
{
    %1
    %2
    mul_dint
}

overload TIME(TIME,REAL)
inline
{
    %1
    dint_to_real
    %2
    mul_real
    real_to_dint
}

overload TIME(TIME,LREAL)
inline
{
    %1
    dint_to_lreal
    %2
    mul_lreal
    lreal_to_dint
}

END_FUNCTION

(* ---- MUX.st ---- *)
FUNCTION MUX : ANY
VAR_INPUT
   K : ANY_INT;
   IN0: ANY;
END_VAR
VAR_IN_EXT
   IN1: ANY;
END_VAR

(* 1 bit *)
overload BOOL  (INT|DINT to INT, BOOL,   ...) inline{ STDLIB(mux_bit) }

(* 8 bit *)
overload BYTE  (INT|DINT to INT, BYTE,   ...) inline{ STDLIB(mux_byte) }

(* 16 bit *)
overload INT   (INT|DINT to INT, INT,    ...) inline{ STDLIB(mux_int) }
overload WORD  (INT|DINT to INT, WORD,   ...) inline{ STDLIB(mux_int) }

(* 32 bit *)
overload DINT  (INT|DINT to INT, DINT,   ...) inline{ STDLIB(mux_dint) }
overload DWORD (INT|DINT to INT, DWORD,  ...) inline{ STDLIB(mux_dint) }
overload TIME  (INT|DINT to INT, TIME,   ...) inline{ STDLIB(mux_dint) }
overload REAL  (INT|DINT to INT, REAL,   ...) inline{ STDLIB(mux_dint) }

(* 64 bit *)
overload LREAL (INT|DINT to INT, LREAL,  ...) inline{ STDLIB(mux_64bit) }

(* string *)
overload STRING(INT|DINT to INT, STRING, ...) inline{ STDLIB(mux_string) }

END_FUNCTION

(* ---- ne.st ---- *)
(*[[
    UserURL= "ATCMfile:NE.htm"
]]*)

FUNCTION NE : BOOL
VAR_INPUT
    IN1 : ANY_ELEMENTARY;
    IN2 : ANY_ELEMENTARY;
END_VAR

inline <>

END_FUNCTION

(* ---- not.st ---- *)
(*[[
    UserURL= "ATCMfile:NOT.htm"
]]*)

FUNCTION NOT : ANY_BIT
VAR_INPUT
    IN : ANY_BIT;
END_VAR

inline NOT

END_FUNCTION

(* ---- or.st ---- *)
(*[[
    UserURL= "ATCMfile:OR.htm"
]]*)

FUNCTION OR : ANY_BIT
VAR_INPUT
    IN1 : ANY_BIT;
END_VAR
VAR_IN_EXT
    IN2 : ANY_BIT;
END_VAR

inline OR

END_FUNCTION

(* ---- real_to_bool.st ---- *)
(*[[
    UserURL= "ATCMfile:REAL_TO_BOOL.htm"
]]*)

FUNCTION REAL_TO_BOOL : BOOL
VAR_INPUT
    IN : REAL;
END_VAR

inline{VMOP}

END_FUNCTION

(* ---- real_to_byte.st ---- *)
(*[[
    UserURL= "ATCMfile:REAL_TO_BYTE.htm"
]]*)

FUNCTION REAL_TO_BYTE : BYTE
VAR_INPUT
    IN : REAL;
END_VAR

inline{VMOP}

END_FUNCTION

(* ---- real_to_dint.st ---- *)
(*[[
    UserURL= "ATCMfile:REAL_TO_DINT.htm"
]]*)

FUNCTION REAL_TO_DINT : DINT
VAR_INPUT
    IN : REAL;
END_VAR

inline{VMOP}

END_FUNCTION

(* ---- real_to_dword.st ---- *)
(*[[
    UserURL= "ATCMfile:REAL_TO_DWORD.htm"
]]*)

FUNCTION REAL_TO_DWORD : DWORD
VAR_INPUT
    IN : REAL;
END_VAR

inline{VMOP}

END_FUNCTION

(* ---- real_to_int.st ---- *)
(*[[
    UserURL= "ATCMfile:REAL_TO_INT.htm"
]]*)

FUNCTION REAL_TO_INT : INT
VAR_INPUT
    IN : REAL;
END_VAR

inline{VMOP}

END_FUNCTION

(* ---- real_to_lint.st ---- *)
(*[[
    UserURL= "ATCMfile:REAL_TO_LINT.htm"
]]*)

FUNCTION REAL_TO_LINT : LINT
VAR_INPUT
    IN : REAL;
END_VAR

inline{VMOP(not_yet_implem)}

END_FUNCTION

(* ---- real_to_lreal.st ---- *)
(*[[
    UserURL= "ATCMfile:REAL_TO_LREAL.htm"
]]*)

FUNCTION REAL_TO_LREAL : LREAL
VAR_INPUT
    IN : REAL;
END_VAR

inline{VMOP}

END_FUNCTION

(* ---- real_to_lword.st ---- *)
(*[[
    UserURL= "ATCMfile:REAL_TO_LWORD.htm"
]]*)

FUNCTION REAL_TO_LWORD : LWORD
VAR_INPUT
    IN : REAL;
END_VAR

inline{VMOP(not_yet_implem)}

END_FUNCTION

(* ---- real_to_string.st ---- *)
(*[[
    UserURL= "ATCMfile:REAL_TO_STRING.htm"
]]*)

FUNCTION REAL_TO_STRING : STRING
VAR_INPUT
    IN : REAL;
END_VAR

inline{ STDLIB(real_to_string) }

END_FUNCTION

(* ---- real_to_time.st ---- *)
(*[[
    UserURL= "ATCMfile:REAL_TO_TIME.htm"
]]*)

FUNCTION REAL_TO_TIME : TIME
VAR_INPUT
    IN : REAL;
END_VAR

inline
{
    %1
    real_to_dint
}

END_FUNCTION

(* ---- real_to_udint.st ---- *)
(*[[
    UserURL= "ATCMfile:REAL_TO_UDINT.htm"
]]*)
FUNCTION REAL_TO_UDINT : UDINT
VAR_INPUT
    IN : REAL;
END_VAR

inline{ VMOP }

END_FUNCTION

(* ---- real_to_uint.st ---- *)
(*[[
    UserURL= "ATCMfile:REAL_TO_UINT.htm"
]]*)
FUNCTION REAL_TO_UINT : UINT
VAR_INPUT
    IN : REAL;
END_VAR

inline{ VMOP }

END_FUNCTION

(* ---- real_to_word.st ---- *)
(*[[
    UserURL= "ATCMfile:REAL_TO_WORD.htm"
]]*)

FUNCTION REAL_TO_WORD : WORD
VAR_INPUT
    IN : REAL;
END_VAR

inline{VMOP}

END_FUNCTION

(* ---- REPLACE.st ---- *)
FUNCTION REPLACE : ANY_STRING
VAR_INPUT
    IN1 : ANY_STRING;
    IN2 : ANY_STRING;
    L : ANY_INT;
    P : ANY_INT;
END_VAR

overload STRING(STRING,STRING, INT,INT)                  inline{ STDLIB(ReplaceString_int) }
overload STRING(STRING,STRING, DINT to INT ,DINT to INT) inline{ STDLIB(ReplaceString_int) }

END_FUNCTION

(* ---- RIGHT.st ---- *)
FUNCTION RIGHT : ANY_STRING
VAR_INPUT
    IN : ANY_STRING;
    L : ANY_INT;
END_VAR

overload STRING(STRING,         INT) inline{ STDLIB(RightString_int) }
overload STRING(STRING, DINT to INT) inline{ STDLIB(RightString_int) }

END_FUNCTION

(* ---- ROL.st ---- *)
FUNCTION ROL : any_bit
VAR_INPUT
    IN : any_bit;
    N  : any_int;
END_VAR

(* we do not support DINT as second param *)
(*
overload bool(bool,dint)
inline
{
    %1
    %2
    dint_to_int
    rol_bool
}
overload byte(byte,dint)
inline
{
    %1
    %2
    dint_to_int
    rol_byte
}
overload word(word,dint)
inline
{
    %1
    %2
    dint_to_int
    rol_word
}
overload dword(dword,dint)
inline
{
    %1
    %2
    dint_to_int
    rol_dword
}
*)

overload bool(bool,int)   inline{ VMOP(rol_bool) }
overload byte(byte,int)   inline{ VMOP(rol_byte) }
overload word(word,int)   inline{ VMOP(rol_word) }
overload dword(dword,int) inline{ VMOP(rol_dword) }

(*
overload LWORD(LWORD,INT) inline{}
overload LWORD(LWORD,DINT) inline{}
*)
END_FUNCTION

(* ---- ROR.st ---- *)
FUNCTION ROR : any_bit
VAR_INPUT
    IN : any_bit;
    N  : any_int;
END_VAR

(* we do not support DINT as second param *)
(*
overload bool(bool,dint)
inline
{
    %1
    %2
    dint_to_int
    ror_bool
}
overload byte(byte,dint)
inline
{
    %1
    %2
    dint_to_int
    ror_byte
}
overload word(word,dint)
inline
{
    %1
    %2
    dint_to_int
    ror_word
}
overload dword(dword,dint)
inline
{
    %1
    %2
    dint_to_int
    ror_dword
}
*)

overload bool(bool,int)   inline{ VMOP(ror_bool) }
overload byte(byte,int)   inline{ VMOP(ror_byte) }
overload word(word,int)   inline{ VMOP(ror_word) }
overload dword(dword,int) inline{ VMOP(ror_dword) }

(*
overload LWORD(LWORD,INT) inline{}
overload LWORD(LWORD,DINT) inline{}
*)
END_FUNCTION

(* ---- SEL.st ---- *)
FUNCTION SEL : ANY

VAR_INPUT
    G   : BOOL;
    IN0 : ANY;
    IN1 : ANY;
END_VAR

overload ANY_ELEMENTARY(BOOL,ANY_ELEMENTARY,ANY_ELEMENTARY) inline
{
    %1
    jmpcn L1%u
    %3
    jmp L2%u
:L1%u
    %2
:L2%u
}
END_FUNCTION

(* ---- SHL.st ---- *)
FUNCTION SHL : any_bit
VAR_INPUT
    IN : any_bit;
    N  : any_int;
END_VAR

(* we do not support DINT as second param *)
(*
overload bool(bool,dint)
inline
{
    %1
    %2
    dint_to_int
    shl_bool
}
overload byte(byte,dint)
inline
{
    %1
    %2
    dint_to_int
    shl_byte
}
overload word(word,dint)
inline
{
    %1
    %2
    dint_to_int
    shl_word
}
overload dword(dword,dint)
inline
{
    %1
    %2
    dint_to_int
    shl_dword
}
*)

overload bool(bool,int)   inline{ VMOP(shl_bool) }
overload byte(byte,int)   inline{ VMOP(shl_byte) }
overload word(word,int)   inline{ VMOP(shl_word) }
overload dword(dword,int) inline{ VMOP(shl_dword) }

(*
overload LWORD(LWORD,INT) inline{}
overload LWORD(LWORD,DINT) inline{}
*)
END_FUNCTION

(* ---- SHR.st ---- *)
FUNCTION SHR : any_bit
VAR_INPUT
    IN : any_bit;
    N  : any_int;
END_VAR

(* we do not support DINT as second param *)
(*
overload bool(bool,dint)
inline
{
    %1
    %2
    dint_to_int
    shr_bool
}
overload byte(byte,dint)
inline
{
    %1
    %2
    dint_to_int
    shr_byte
}
overload word(word,dint)
inline
{
    %1
    %2
    dint_to_int
    shr_word
}
overload dword(dword,dint)
inline
{
    %1
    %2
    dint_to_int
    shr_dword
}
*)

overload bool(bool,int)   inline{ VMOP(shr_bool) }
overload byte(byte,int)   inline{ VMOP(shr_byte) }
overload word(word,int)   inline{ VMOP(shr_word) }
overload dword(dword,int) inline{ VMOP(shr_dword) }

(*
overload LWORD(LWORD,INT) inline{}
overload LWORD(LWORD,DINT) inline{}
*)

END_FUNCTION

(* ---- SIN.st ---- *)
FUNCTION SIN : any_real
VAR_INPUT
    IN : any_real;
END_VAR

overload lreal(lreal) inline { STDLIB(sin_lreal) }
overload real(real)   inline { STDLIB(sin_real) }

END_FUNCTION

(* ---- sqrt.st ---- *)
FUNCTION SQRT : any_real
VAR_INPUT
    IN : any_real;
END_VAR

overload lreal(lreal) inline { STDLIB(sqrt_lreal) }
overload real(real) inline   { STDLIB(sqrt_real) }

END_FUNCTION

(* ---- string_to_bool.st ---- *)
(*[[
    UserURL= "ATCMfile:WSTRING_TO_BOOL.htm"
]]*)

FUNCTION STRING_TO_BOOL : BOOL
VAR_INPUT
    IN : STRING;
END_VAR

inline { STDLIB(string_to_bool) }

END_FUNCTION

(* ---- string_to_byte.st ---- *)
(*[[
    UserURL= "ATCMfile:STRING_TO_BYTE.htm"
]]*)

FUNCTION STRING_TO_BYTE : BYTE
VAR_INPUT
    IN : STRING;
END_VAR

inline{ STDLIB(string_to_byte) }

END_FUNCTION

(* ---- string_to_date.st ---- *)
(*[[
    UserURL= "ATCMfile:STRING_TO_DATE.htm"
]]*)

FUNCTION STRING_TO_DATE : DATE
VAR_INPUT
    IN : STRING;
END_VAR

inline{ STDLIB(string_to_date) }

END_FUNCTION

(* ---- string_to_dint.st ---- *)
(*[[
    UserURL= "ATCMfile:WSTRING_TO_DINT.htm"
]]*)

FUNCTION STRING_TO_DINT : DINT
VAR_INPUT
    IN : STRING;
END_VAR

inline{ STDLIB(string_to_dint) }

END_FUNCTION

(* ---- string_to_dt.st ---- *)
(*[[
    UserURL= "ATCMfile:WSTRING_TO_DT.htm"
]]*)

FUNCTION STRING_TO_DT : DT
VAR_INPUT
    IN : STRING;
END_VAR

inline{VMOP(not_yet_implem)}

END_FUNCTION

(* ---- string_to_dword.st ---- *)
(*[[
    UserURL= "ATCMfile:WSTRING_TO_DWORD.htm"
]]*)

FUNCTION STRING_TO_DWORD : DWORD
VAR_INPUT
    IN : STRING;
END_VAR

inline{ STDLIB(string_to_dword) }

END_FUNCTION

(* ---- string_to_int.st ---- *)
(*[[
    UserURL= "ATCMfile:WSTRING_TO_LINT.htm"
]]*)

FUNCTION STRING_TO_INT : INT
VAR_INPUT
    IN : STRING;
END_VAR

inline{ STDLIB(string_to_int) }

END_FUNCTION

(* ---- string_to_lint.st ---- *)
(*[[
    UserURL= "ATCMfile:WSTRING_TO_LINT.htm"
]]*)

FUNCTION STRING_TO_LINT : LINT
VAR_INPUT
    IN : STRING;
END_VAR

inline{VMOP(not_yet_implem)}

END_FUNCTION

(* ---- string_to_lreal.st ---- *)
(*[[
    UserURL= "ATCMfile:WSTRING_TO_LREAL.htm"
]]*)

FUNCTION STRING_TO_LREAL : LREAL
VAR_INPUT
    IN : STRING;
END_VAR

inline{ STDLIB(string_to_lreal) }

END_FUNCTION

(* ---- string_to_lword.st ---- *)
(*[[
    UserURL= "ATCMfile:WSTRING_TO_LWORD.htm"
]]*)

FUNCTION STRING_TO_LWORD : LWORD
VAR_INPUT
    IN : STRING;
END_VAR

inline{VMOP(not_yet_implem)}

END_FUNCTION

(* ---- string_to_real.st ---- *)
(*[[
    UserURL= "ATCMfile:WSTRING_TO_LREAL.htm"
]]*)

FUNCTION STRING_TO_REAL : REAL
VAR_INPUT
    IN : STRING;
END_VAR

inline{ STDLIB(string_to_real) }
END_FUNCTION

(* ---- string_to_time.st ---- *)
(*[[
    UserURL= "ATCMfile:WSTRING_TO_TIME.htm"
]]*)

FUNCTION STRING_TO_TIME : TIME
VAR_INPUT
    IN : STRING;
END_VAR

inline{ STDLIB(string_to_time) }

END_FUNCTION

(* ---- string_to_tod.st ---- *)
(*[[
    UserURL= "ATCMfile:WSTRING_TO_TOD.htm"
]]*)

FUNCTION STRING_TO_TOD : TOD
VAR_INPUT
    IN : STRING;
END_VAR

inline{VMOP(not_yet_implem)}

END_FUNCTION

(* ---- string_to_udint.st ---- *)
(*[[
    UserURL= "ATCMfile:STRING_TO_UDINT.htm"
]]*)
FUNCTION STRING_TO_UDINT : UDINT
VAR_INPUT
    IN : STRING;
END_VAR

inline{ STDLIB(string_to_dword) }

END_FUNCTION

(* ---- string_to_uint.st ---- *)
(*[[
    UserURL= "ATCMfile:STRING_TO_UINT.htm"
]]*)
FUNCTION STRING_TO_UINT : UINT
VAR_INPUT
    IN : STRING;
END_VAR

inline{ STDLIB(string_to_word) }

END_FUNCTION

(* ---- string_to_word.st ---- *)
(*[[
    UserURL= "ATCMfile:WSTRING_TO_WORD.htm"
]]*)

FUNCTION STRING_TO_WORD : WORD
VAR_INPUT
    IN : STRING;
END_VAR

inline{ STDLIB(string_to_word) }

END_FUNCTION

(* ---- sub.st ---- *)
(*[[
    UserURL= "ATCMfile:SUB.htm"
]]*)

FUNCTION SUB : ANY_MAGNITUDE
VAR_INPUT
    IN1: ANY_MAGNITUDE;
    IN2: ANY_MAGNITUDE;
END_VAR

inline -

END_FUNCTION

(* ---- sub_time.st ---- *)
(*[[
    UserURL= "ATCMfile:SUB_TIME.htm"
]]*)

FUNCTION SUB_TIME : TIME
VAR_INPUT
    IN1 : TIME;
    IN2 : TIME;
END_VAR

inline -

END_FUNCTION

(* ---- TAN.st ---- *)
FUNCTION TAN : any_real
VAR_INPUT
    IN : any_real;
END_VAR

overload lreal(lreal) inline { STDLIB(tan_lreal) }
overload real(real)   inline { STDLIB(tan_real) }

END_FUNCTION

(* ---- time_to_dint.st ---- *)
(*[[
    UserURL= "ATCMfile:TIME_TO_DINT.htm"
]]*)

FUNCTION TIME_TO_DINT : DINT
VAR_INPUT
    IN : TIME;
END_VAR

inline { %1 }

END_FUNCTION

(* ---- time_to_dt.st ---- *)
(*[[
    UserURL= "ATCMfile:TIME_TO_DT.htm"
]]*)

FUNCTION TIME_TO_DT : DT
VAR_INPUT
    IN : TIME;
END_VAR

inline{%1}

END_FUNCTION

(* ---- time_to_int.st ---- *)
(*[[
    UserURL= "ATCMfile:TIME_TO_LINT.htm"
]]*)

FUNCTION TIME_TO_INT : INT
VAR_INPUT
    IN : TIME;
END_VAR

inline
{
    %1
    dint_to_int
}

END_FUNCTION

(* ---- time_to_lint.st ---- *)
(*[[
    UserURL= "ATCMfile:TIME_TO_LINT.htm"
]]*)

FUNCTION TIME_TO_LINT : LINT
VAR_INPUT
    IN : TIME;
END_VAR

inline{%1}

END_FUNCTION

(* ---- time_to_lreal.st ---- *)
(*[[
    UserURL= "ATCMfile:TIME_TO_LREAL.htm"
]]*)

FUNCTION TIME_TO_LREAL : LREAL
VAR_INPUT
    IN : TIME;
END_VAR

inline
{
    %1
    dint_to_lreal
}

END_FUNCTION

(* ---- time_to_real.st ---- *)
(*[[
    UserURL= "ATCMfile:TIME_TO_LREAL.htm"
]]*)

FUNCTION TIME_TO_REAL : REAL
VAR_INPUT
    IN : TIME;
END_VAR

inline
{
    %1
    dint_to_real
}

END_FUNCTION

(* ---- time_to_string.st ---- *)
(*[[
    UserURL= "ATCMfile:TIME_TO_WSTRING.htm"
]]*)

FUNCTION TIME_TO_STRING : STRING
VAR_INPUT
   IN : TIME;
END_VAR

inline{ STDLIB(time32_to_string) }

END_FUNCTION

(* ---- tod_to_string.st ---- *)
(*[[
    UserURL= "ATCMfile:TOD_TO_STRING.htm"
]]*)

FUNCTION TOD_TO_STRING : STRING
VAR_INPUT
    IN : TOD;
END_VAR

inline{ STDLIB(not yet implented) }

END_FUNCTION

(* ---- tod_to_time.st ---- *)
(*[[
    UserURL= "ATCMfile:TOD_TO_TIME.htm"
]]*)

FUNCTION TOD_TO_TIME : TIME
VAR_INPUT
    IN : TOD;
END_VAR

inline{(long)%1}

END_FUNCTION

(* ---- trunc.st ---- *)
(*[[
    UserURL= "ATCMfile:TRUNC.htm"
]]*)

FUNCTION TRUNC : ANY_INT
VAR_INPUT
    IN : ANY_REAL;
END_VAR

overload DINT        (REAL)  inline{ STDLIB(Trunc_real_dint) }
overload DINT        (LREAL) inline{ STDLIB(Trunc_lreal_dint) }
overload DINT to INT (REAL)  inline{ STDLIB(Trunc_real_dint) }
overload DINT to INT (LREAL) inline{ STDLIB(Trunc_lreal_dint) }

END_FUNCTION

(* ---- udint_to_bool.st ---- *)
(*[[
    UserURL= "ATCMfile:UDINT_TO_BOOL.htm"
]]*)
FUNCTION UDINT_TO_BOOL : BOOL
VAR_INPUT
    IN : UDINT;
END_VAR

inline{ VMOP }

END_FUNCTION

(* ---- udint_to_byte.st ---- *)
(*[[
    UserURL= "ATCMfile:UDINT_TO_BYTE.htm"
]]*)
FUNCTION UDINT_TO_BYTE : BYTE
VAR_INPUT
    IN : UDINT;
END_VAR

inline{ VMOP }

END_FUNCTION

(* ---- udint_to_dint.st ---- *)
(*[[
    UserURL= "ATCMfile:UDINT_TO_DINT.htm"
]]*)
FUNCTION UDINT_TO_DINT : DINT
VAR_INPUT
    IN : UDINT;
END_VAR

inline{NOOP}

END_FUNCTION

(* ---- udint_to_dword.st ---- *)
(*[[
    UserURL= "ATCMfile:UDINT_TO_DWORD.htm"
]]*)
FUNCTION UDINT_TO_DWORD : DWORD
VAR_INPUT
    IN : UDINT;
END_VAR

inline{NOOP}

END_FUNCTION

(* ---- udint_to_int.st ---- *)
(*[[
    UserURL= "ATCMfile:UDINT_TO_INT.htm"
]]*)
FUNCTION UDINT_TO_INT : INT
VAR_INPUT
    IN : UDINT;
END_VAR

inline{ VMOP }

END_FUNCTION

(* ---- udint_to_lreal.st ---- *)
(*[[
    UserURL= "ATCMfile:UDINT_TO_LREAL.htm"
]]*)
FUNCTION UDINT_TO_LREAL : LREAL
VAR_INPUT
    IN : UDINT;
END_VAR

inline{ VMOP }

END_FUNCTION

(* ---- udint_to_real.st ---- *)
(*[[
    UserURL= "ATCMfile:UDINT_TO_REAL.htm"
]]*)
FUNCTION UDINT_TO_REAL : REAL
VAR_INPUT
    IN : UDINT;
END_VAR

inline{ VMOP }

END_FUNCTION

(* ---- udint_to_string.st ---- *)
(*[[
    UserURL= "ATCMfile:UDINT_TO_STRING.htm"
]]*)
FUNCTION UDINT_TO_STRING : STRING
VAR_INPUT
    IN : UDINT;
END_VAR

inline{ STDLIB(dword_to_string) }

END_FUNCTION

(* ---- udint_to_word.st ---- *)
(*[[
    UserURL= "ATCMfile:UDINT_TO_WORD.htm"
]]*)
FUNCTION UDINT_TO_WORD : WORD
VAR_INPUT
    IN : UDINT;
END_VAR

inline{ VMOP }

END_FUNCTION

(* ---- uint_to_bool.st ---- *)
(*[[
    UserURL= "ATCMfile:UINT_TO_BOOL.htm"
]]*)
FUNCTION UINT_TO_BOOL : BOOL
VAR_INPUT
    IN : UINT;
END_VAR

inline{ VMOP }

END_FUNCTION

(* ---- uint_to_byte.st ---- *)
(*[[
    UserURL= "ATCMfile:UINT_TO_BYTE.htm"
]]*)
FUNCTION UINT_TO_BYTE : BYTE
VAR_INPUT
    IN : UINT;
END_VAR

inline{ VMOP }

END_FUNCTION

(* ---- uint_to_dint.st ---- *)
(*[[
    UserURL= "ATCMfile:UINT_TO_DINT.htm"
]]*)
FUNCTION UINT_TO_DINT : DINT
VAR_INPUT
    IN : UINT;
END_VAR

inline{ VMOP }

END_FUNCTION

(* ---- uint_to_dword.st ---- *)
(*[[
    UserURL= "ATCMfile:UINT_TO_DWORD.htm"
]]*)
FUNCTION UINT_TO_DWORD : DWORD
VAR_INPUT
    IN : UINT;
END_VAR

inline{ VMOP }

END_FUNCTION

(* ---- uint_to_int.st ---- *)
(*[[
    UserURL= "ATCMfile:UINT_TO_INT.htm"
]]*)
FUNCTION UINT_TO_INT : INT
VAR_INPUT
    IN : UINT;
END_VAR

inline{NOOP}

END_FUNCTION

(* ---- uint_to_lreal.st ---- *)
(*[[
    UserURL= "ATCMfile:UINT_TO_LREAL.htm"
]]*)
FUNCTION UINT_TO_LREAL : LREAL
VAR_INPUT
    IN : UINT;
END_VAR

inline{ VMOP }

END_FUNCTION

(* ---- uint_to_real.st ---- *)
(*[[
    UserURL= "ATCMfile:UINT_TO_REAL.htm"
]]*)
FUNCTION UINT_TO_REAL : REAL
VAR_INPUT
    IN : UINT;
END_VAR

inline{ VMOP }

END_FUNCTION

(* ---- uint_to_string.st ---- *)
(*[[
    UserURL= "ATCMfile:UINT_TO_STRING.htm"
]]*)
FUNCTION UINT_TO_STRING : STRING
VAR_INPUT
    IN : UINT;
END_VAR

inline{ STDLIB(word_to_string) }

END_FUNCTION

(* ---- uint_to_word.st ---- *)
(*[[
    UserURL= "ATCMfile:UINT_TO_WORD.htm"
]]*)
FUNCTION UINT_TO_WORD : WORD
VAR_INPUT
    IN : UINT;
END_VAR

inline{NOOP}

END_FUNCTION

(* ---- word_string.st ---- *)
(*[[
    UserURL= "ATCMfile:WORD_TO_WSTRING.htm"
]]*)

FUNCTION WORD_TO_STRING : STRING
VAR_INPUT
    IN : WORD;
END_VAR

inline{VMOP}

END_FUNCTION

(* ---- word_to_bool.st ---- *)
(*[[
    UserURL= "ATCMfile:WORD_TO_BOOL.htm"
]]*)

FUNCTION WORD_TO_BOOL : BOOL
VAR_INPUT
    IN : WORD;
END_VAR

inline{VMOP}

END_FUNCTION

(* ---- word_to_byte.st ---- *)
(*[[
    UserURL= "ATCMfile:WORD_TO_BYTE.htm"
]]*)

FUNCTION WORD_TO_BYTE : BYTE
VAR_INPUT
    IN : WORD;
END_VAR

inline{VMOP}

END_FUNCTION

(* ---- word_to_dint.st ---- *)
(*[[
    UserURL= "ATCMfile:WORD_TO_DINT.htm"
]]*)

FUNCTION WORD_TO_DINT : DINT
VAR_INPUT
    IN : WORD;
END_VAR

inline{VMOP(word_to_dword)}

END_FUNCTION

(* ---- word_to_dword.st ---- *)
(*[[
    UserURL= "ATCMfile:WORD_TO_DWORD.htm"
]]*)

FUNCTION WORD_TO_DWORD : DWORD
VAR_INPUT
    IN : WORD;
END_VAR

inline{VMOP}

END_FUNCTION

(* ---- word_to_int.st ---- *)
(*[[
    UserURL= "ATCMfile:WORD_TO_INT.htm"
]]*)

FUNCTION WORD_TO_INT : INT
VAR_INPUT
    IN : WORD;
END_VAR

inline{NOOP}

END_FUNCTION

(* ---- word_to_lint.st ---- *)
(*[[
    UserURL= "ATCMfile:WORD_TO_LINT.htm"
]]*)

FUNCTION WORD_TO_LINT : LINT
VAR_INPUT
    IN : WORD;
END_VAR

inline{VMOP(not_yet_implem)}

END_FUNCTION

(* ---- word_to_lreal.st ---- *)
(*[[
    UserURL= "ATCMfile:WORD_TO_LREAL.htm"
]]*)

FUNCTION WORD_TO_LREAL : LREAL
VAR_INPUT
    IN : WORD;
END_VAR

inline{VMOP}

END_FUNCTION

(* ---- word_to_lword.st ---- *)
(*[[
    UserURL= "ATCMfile:WORD_TO_LWORD.htm"
]]*)

FUNCTION WORD_TO_LWORD : LWORD
VAR_INPUT
    IN : WORD;
END_VAR

inline{VMOP(not_yet_implem)}

END_FUNCTION

(* ---- word_to_real.st ---- *)
(*[[
    UserURL= "ATCMfile:WORD_TO_LREAL.htm"
]]*)

FUNCTION WORD_TO_REAL : REAL
VAR_INPUT
    IN : WORD;
END_VAR

inline{VMOP}

END_FUNCTION

(* ---- word_to_string.st ---- *)
(*[[
    UserURL= "ATCMfile:WORD_TO_WSTRING.htm"
]]*)

FUNCTION WORD_TO_STRING : STRING
VAR_INPUT
    IN : WORD;
END_VAR

inline{ STDLIB(word_to_string) }

END_FUNCTION

(* ---- word_to_udint.st ---- *)
(*[[
    UserURL= "ATCMfile:WORD_TO_UDINT.htm"
]]*)
FUNCTION WORD_TO_UDINT : UDINT
VAR_INPUT
    IN : WORD;
END_VAR

inline{ VMOP }

END_FUNCTION

(* ---- word_to_uint.st ---- *)
(*[[
    UserURL= "ATCMfile:WORD_TO_UINT.htm"
]]*)
FUNCTION WORD_TO_UINT : UINT
VAR_INPUT
    IN : WORD;
END_VAR

inline{NOOP}

END_FUNCTION

(* ---- xor.st ---- *)
(*[[
    UserURL= "ATCMfile:XOR.htm"
]]*)

FUNCTION XOR : ANY_BIT
VAR_INPUT
    IN1 : ANY_BIT;
END_VAR
VAR_IN_EXT
    IN2 : ANY_BIT;
END_VAR

inline XOR

END_FUNCTION

(* ---- ctd.st ---- *)
(*[[
    UserURL= "ATCMfile:TOF.htm"
]]*)
(*
 *  IEC-1131-3 Standard Functionblock CTD for data type INT
 *  Purpose: Down Counter
 *)
FUNCTION_BLOCK CTD
VAR_INPUT  (* Inputs *)
    CD         : BOOL R_EDGE; (* count down if rising edge     *)
    LD         : BOOL;        (* if true, copy PV to CV        *)
    PV         : INT;         (* start value                   *)
END_VAR
VAR_OUTPUT (* Outputs *)
    Q          : BOOL;        (* TRUE if CV <= 0               *)
    CV         : INT;         (* counter output                *)
END_VAR

inline { STDLIB(ctd) }

END_FUNCTION_BLOCK

(* ---- ctu.st ---- *)
(*[[
    UserURL= "ATCMfile:TON.htm"
]]*)
(*
 *  IEC-1131-3 Standard Functionblock CTU for data type INT
 *  Purpose: Up Counter
 *)
FUNCTION_BLOCK CTU
VAR_INPUT (* Inputs *)
    CU         : BOOL R_EDGE; (* count up if rising edge *)
    R          : BOOL;        (* if true,  CV to zero    *)
    PV         : INT;         (* end value               *)
END_VAR
VAR_OUTPUT (* Outputs *)
    Q          : BOOL;        (* TRUE if CV >= PV        *)
    CV         : INT;         (* counter output          *)
END_VAR

inline { STDLIB(ctu) }

END_FUNCTION_BLOCK

(* ---- ctud.st ---- *)
(*[[
    UserURL= "ATCMfile:TP.htm"
]]*)
(*
 *  IEC-1131-3 Standard Functionblock CTUD for data type DINT
 *  Purpose: Up/Down Counter
 *)
FUNCTION_BLOCK CTUD
VAR_INPUT (* Inputs *)
    CU         : BOOL R_EDGE; (* count up if rising edge   *)
    CD         : BOOL R_EDGE; (* count down if rising edge *)
    R          : BOOL;        (* Reset, set CV to 0        *)
    LD         : BOOL;        (* if true, copy PV to CV    *)
    PV         : INT;         (* start value               *)
END_VAR
VAR_OUTPUT (* Outputs *)
    QU         : BOOL;        (* TRUE if CV >= PV          *)
    QD         : BOOL;        (* TRUE if CV <= 0           *)
    CV         : INT;         (* counter output            *)
END_VAR

inline { STDLIB(ctud) }

END_FUNCTION_BLOCK

(* ---- f_trig.st ---- *)
FUNCTION_BLOCK F_TRIG
VAR_INPUT
	CLK: BOOL;
END_VAR
VAR_OUTPUT
	Q: BOOL;
END_VAR
VAR
	M: BOOL := TRUE;
END_VAR

(*
Q := NOT CLK AND NOT M;
M := NOT CLK;
*)

inline { STDLIB(f_trig) }

END_FUNCTION_BLOCK

(* ---- r_trig.st ---- *)
FUNCTION_BLOCK R_TRIG
VAR_INPUT
	CLK: BOOL;
END_VAR
VAR_OUTPUT
	Q: BOOL;
END_VAR
VAR
	M: BOOL := FALSE;
END_VAR

(*
Q := CLK AND NOT M;
M := CLK;
*)

inline { STDLIB(r_trig) }

END_FUNCTION_BLOCK

(* ---- rs.st ---- *)
FUNCTION_BLOCK RS
VAR_INPUT
   S  : BOOL;
   R1 : BOOL;
END_VAR
VAR_OUTPUT
   Q1 : BOOL;
END_VAR

(*
 Q1 := NOT R1 AND (S OR Q1);
*)
inline { STDLIB(rs) }

END_FUNCTION_BLOCK

(* ---- sr.st ---- *)
FUNCTION_BLOCK SR
VAR_INPUT
   S1 : BOOL;
   R  : BOOL;
END_VAR
VAR_OUTPUT
   Q1 : BOOL;
END_VAR

(*
  Q1 := (NOT R AND Q1) OR S1;
*)
inline { STDLIB(SR) }

END_FUNCTION_BLOCK

(* ---- tof.st ---- *)
(*[[
    UserURL= "ATCMfile:TOF.htm"
]]*)

FUNCTION_BLOCK TOF

VAR_INPUT   (* Inputs *)
    IN : BOOL := FALSE; (* Input        *)
    PT : TIME := T#0s;  (* Preset time  *)
END_VAR

VAR_OUTPUT  (* Outputs *)
    Q  : BOOL := FALSE; (* FALSE if ET >= PT *)
    ET : TIME := T#0s; (* Elapsed time      *)
END_VAR

VAR NON_RETAIN
    StartTime : TIME;
    State : INT := 0;
END_VAR

VAR
    M         : BOOL := FALSE;
END_VAR

inline { STDLIB(tof) }

END_FUNCTION_BLOCK

(* ---- ton.st ---- *)
(*[[
   UserURL= "ATCMfile:TON.htm"
]]*)

FUNCTION_BLOCK TON

VAR_INPUT   (* Inputs *)
    IN : BOOL := FALSE; (* Input        *)
    PT : TIME := T#0s;  (* Preset time 	*)
END_VAR

VAR_OUTPUT  (* Outputs *)
    Q  : BOOL := FALSE; (* TRUE if ET >= PT *)
    ET : TIME := T#0s;  (* Elapsed time     *)
END_VAR

VAR NON_RETAIN
    StartTime : TIME;
    State : INT := 0;
END_VAR

VAR
    M         : BOOL := FALSE;
END_VAR

inline { STDLIB(ton) }

END_FUNCTION_BLOCK

(* ---- tp.st ---- *)
(*[[
    UserURL= "ATCMfile:TP.htm"
]]*)

FUNCTION_BLOCK TP

VAR_INPUT   (* Inputs *)
    IN : BOOL := FALSE; (* Input       *)
    PT : TIME := T#0s;  (* Preset time *)
END_VAR

VAR_OUTPUT  (* Outputs *)
    Q  : BOOL := FALSE; (* FALSE if ET >= PT    *)
    ET : TIME := T#0s;  (* Elapsed time         *)
END_VAR

VAR NON_RETAIN
    StartTime : TIME;
    State     : INT := 0;
END_VAR

VAR
    M         : BOOL := FALSE;
END_VAR

inline { STDLIB(tp) }

END_FUNCTION_BLOCK
